// Mitsubishi GX Works2 project: Class8_Ex02(컨베이어&실린더)   PLC: Q03UD

PROGRAM MAIN
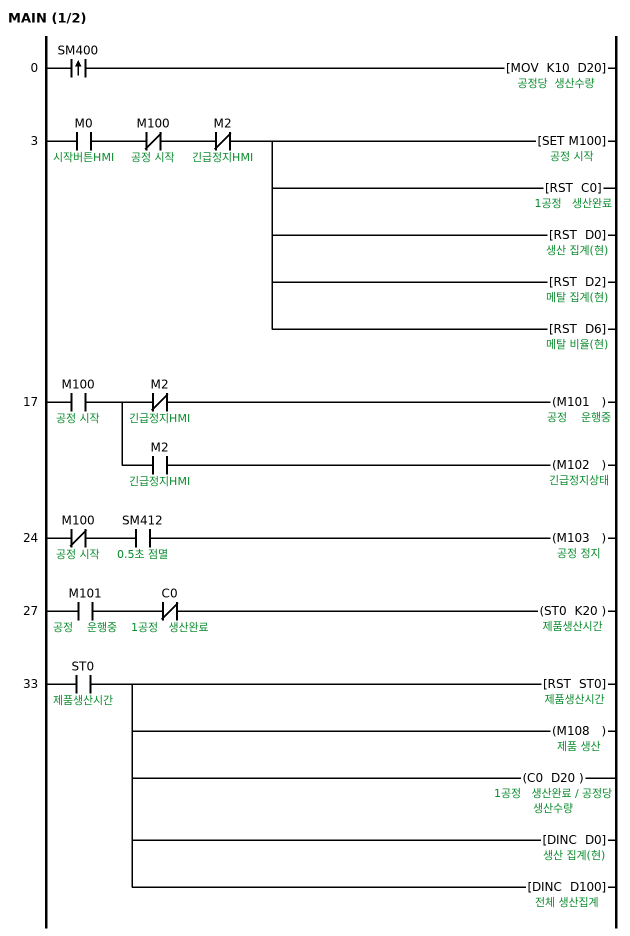
0     LDP     SM400
      MOV     K10 D20  ; 공정당  생산수량
3     LD      M0  ; 시작버튼HMI
      ANI     M100  ; 공정 시작
      ANI     M2  ; 긴급정지HMI
      SET     M100  ; 공정 시작
      RST     C0  ; 1공정   생산완료
      RST     D0  ; 생산 집계(현)
      RST     D2  ; 메탈 집계(현)
      RST     D6  ; 메탈 비율(현)
17    LD      M100  ; 공정 시작
      MPS
      ANI     M2  ; 긴급정지HMI
      OUT     M101  ; 공정    운행중
      MPP
      AND     M2  ; 긴급정지HMI
      OUT     M102  ; 긴급정지상태
24    LDI     M100  ; 공정 시작
      AND     SM412  ; 0.5초 점멸
      OUT     M103  ; 공정 정지
27    LD      M101  ; 공정    운행중
      ANI     C0  ; 1공정   생산완료
      OUT     ST0 K20  ; 제품생산시간
33    LD      ST0  ; 제품생산시간
      RST     ST0  ; 제품생산시간
      OUT     M108  ; 제품 생산
      OUT     C0 D20  ; 1공정   생산완료 / 공정당  생산수량
      DINC    D0
      DINC    D100  ; 전체 생산집계
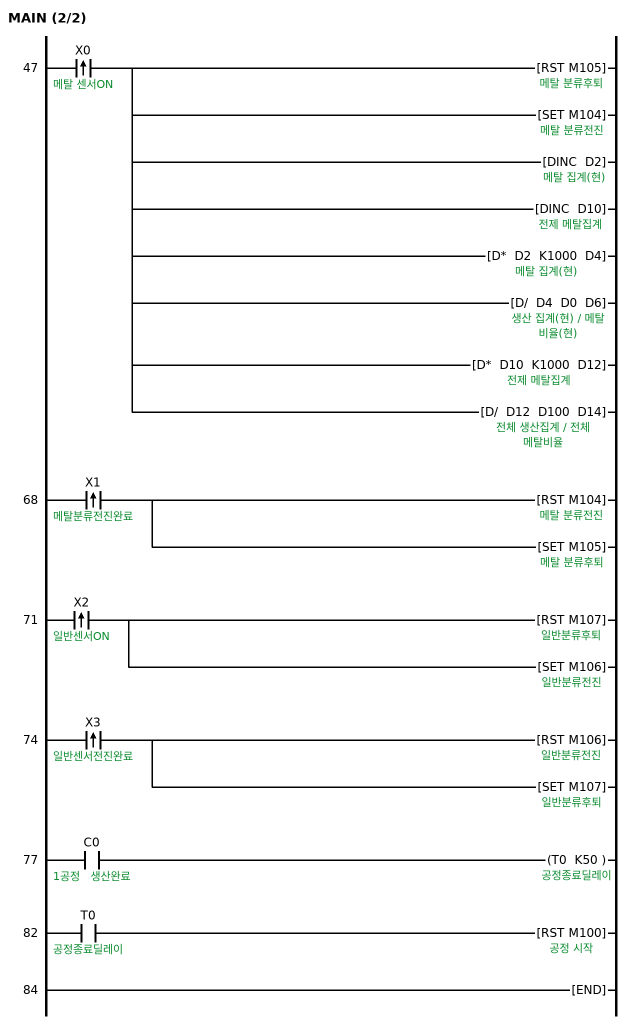
47    LDP     X0  ; 메탈 센서ON
      RST     M105  ; 메탈 분류후퇴
      SET     M104  ; 메탈 분류전진
      DINC    D2
      DINC    D10  ; 전제 메탈집계
      D*      D2 K1000 D4
      D/      D4 D0 D6
      D*      D10 K1000 D12
      D/      D12 D100 D14  ; 전체 메탈비율
68    LDP     X1  ; 메탈분류전진완료
      RST     M104  ; 메탈 분류전진
      SET     M105  ; 메탈 분류후퇴
71    LDP     X2  ; 일반센서ON
      RST     M107  ; 일반분류후퇴
      SET     M106  ; 일반분류전진
74    LDP     X3  ; 일반센서전진완료
      RST     M106  ; 일반분류전진
      SET     M107  ; 일반분류후퇴
77    LD      C0  ; 1공정   생산완료
      OUT     T0 K50  ; 공정종료딜레이
82    LD      T0  ; 공정종료딜레이
      RST     M100  ; 공정 시작
84    END
END_PROGRAM

PROGRAM OUTPUT
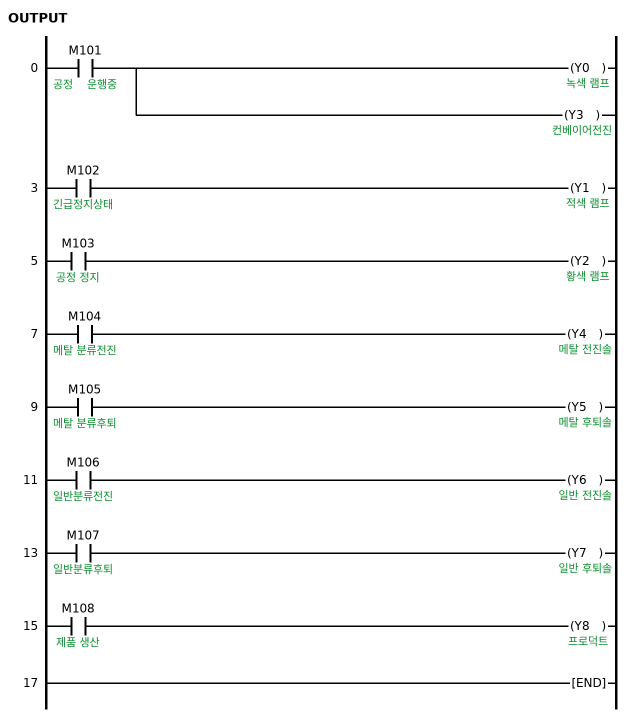
0     LD      M101  ; 공정    운행중
      OUT     Y0  ; 녹색 램프
      OUT     Y3  ; 컨베이어전진
3     LD      M102  ; 긴급정지상태
      OUT     Y1  ; 적색 램프
5     LD      M103  ; 공정 정지
      OUT     Y2  ; 황색 램프
7     LD      M104  ; 메탈 분류전진
      OUT     Y4  ; 메탈 전진솔
9     LD      M105  ; 메탈 분류후퇴
      OUT     Y5  ; 메탈 후퇴솔
11    LD      M106  ; 일반분류전진
      OUT     Y6  ; 일반 전진솔
13    LD      M107  ; 일반분류후퇴
      OUT     Y7  ; 일반 후퇴솔
15    LD      M108  ; 제품 생산
      OUT     Y8  ; 프로덕트
17    END
END_PROGRAM

// device comments not shown above
X4  ; 후퇴리드센서2
X5  ; 정회전신호
X6  ; 역회전신호
X7  ; 비상정지스위치
X8  ; 메탈감지센서
X9  ; 플라스틱감지센서
X10  ; 제품생산시작
Y25  ; 로드 전진1
Y26  ; 로드 후퇴1
Y27  ; 로드전진2
Y28  ; 로드후퇴2
Y29  ; 제품 생산
Y30  ; 컨베이어정회전
Y31  ; 컨베이어역회전
Y32  ; 녹색 램프
Y33  ; 적색 램프
Y34  ; 녹색 램프
Y35  ; 적색 램프
M1  ; 후퇴작동신호1
M3  ; 후퇴작동신호2
M4  ; 정회전ON
M5  ; 역회전ON
M6  ; 제품생산시작
M7  ; 감지중
M8  ; 감지중
M10  ; 시작버튼HMI
M11  ; 긴급정지HMI
T2  ; 3초타이머
T3  ; 0초타이머
